// TIA Portal project "5 Run - 2 Stop For 3 Times" (V16)

(* hardware
DEVICE "S7-1200 station_1"  S7-1200 Station
   slot 0: "Rack_0"  S7-1200 Rack  Rack  V1.0
   slot 1: "PLC_1"  CPU 1212C AC/DC/Rly  6ES7 212-1BE40-0XB0  V4.0
*)

// ===== PLC "PLC_1"  CPU 1212C AC/DC/Rly =====

VAR_GLOBAL   // PLC tag table "Default tag table"
   "start1" AT %I0.2 : Bool;
   "K1" AT %Q0.0 : Bool;
   "stop1" AT %I0.4 : Bool;
   "k2" AT %Q0.1 : Bool;
   "STOP" AT %I0.3 : Bool;
   "T1 tag" AT %M0.0 : Bool;
   "T2 tag" AT %M0.1 : Bool;
   "X" AT %M0.2 : Bool;
   "K3" AT %Q0.2 : Bool;
   "Tag_1" AT %M1.0 : Bool;
   "Tag_2" AT %M1.1 : Bool;
   "Tag_3" AT %M1.2 : Bool;
   "Tag_4" AT %M2.4 : Bool;
   "Tag_5" AT %M7.2 : Bool;
END_VAR

// folder: System blocks/Program resources

DATA_BLOCK "IEC_Counter_0_DB"   // DB1
{ S7_Optimized_Access := 'TRUE' }
AUTHOR : Simatic
FAMILY : IEC
NAME : CNTR
VERSION : 1.0
// stored: InstanceOfName IEC_COUNTER
"IEC_COUNTER"
BEGIN
END_DATA_BLOCK

DATA_BLOCK "T1"   // DB2
{ S7_Optimized_Access := 'TRUE' }
AUTHOR : Simatic
FAMILY : IEC
NAME : IEC_TMR
VERSION : 1.0
// stored: InstanceOfName IEC_TIMER
"IEC_TIMER"
BEGIN
END_DATA_BLOCK

DATA_BLOCK "T2"   // DB3
{ S7_Optimized_Access := 'TRUE' }
AUTHOR : Simatic
FAMILY : IEC
NAME : IEC_TMR
VERSION : 1.0
// stored: InstanceOfName IEC_TIMER
"IEC_TIMER"
BEGIN
END_DATA_BLOCK

// folder: (top level)

ORGANIZATION_BLOCK "Main"   // OB1, LAD, ProgramCycle
TITLE = "Main Program Sweep (Cycle)"
{ S7_Optimized_Access := 'TRUE' }
VERSION : 0.1
   VAR_INPUT
      Initial_Call : Bool;   // Initial call of this OB
      Remanence : Bool;   // =True, if remanent data are available
   END_VAR
   VAR_TEMP   // added for the SCL form of the ladder/FBD networks
      _w1 : Bool;
   END_VAR
BEGIN

REGION Network 1: start
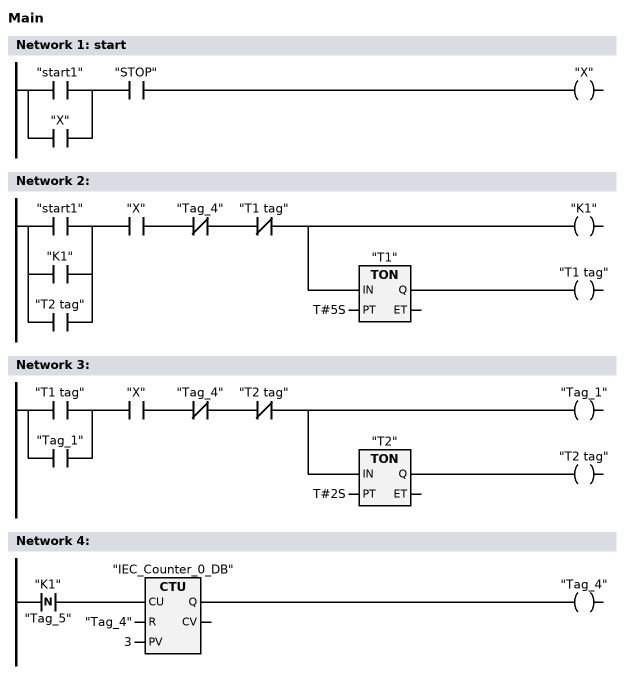
   RUNG wire#powerrail
      Contact( "start1" )
      wire#w1
      Contact( "STOP" )
      Coil( "X" )
   END_RUNG
   RUNG wire#powerrail
      Contact( "X" )
   END_RUNG wire#w1
   // the same network as SCL:
   "X" := ("start1" OR "X") AND "STOP";
END_REGION

REGION Network 2
   "K1" := ("start1" OR "K1" OR "T2 tag") AND "X" AND NOT "Tag_4" AND NOT "T1 tag";
   "T1".TON(IN := "K1", PT := T#5S);
   "T1 tag" := "T1".Q;
END_REGION

REGION Network 3
   "Tag_1" := ("T1 tag" OR "Tag_1") AND "X" AND NOT "Tag_4" AND NOT "T2 tag";
   "T2".TON(IN := "Tag_1", PT := T#2S);
   "T2 tag" := "T2".Q;
END_REGION

REGION Network 4
   #_w1 := NOT "K1" AND "Tag_5";   // falling edge of "K1"
   "Tag_5" := "K1";
   "IEC_Counter_0_DB".CTU(CU := #_w1, R := "Tag_4", PV := 3);
   "Tag_4" := "IEC_Counter_0_DB".Q;
END_REGION
END_ORGANIZATION_BLOCK